PROGRAM F32_InterimPrinter
VAR
END_VAR

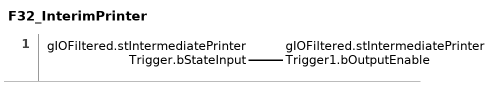
// NETWORK 1
gIOFiltered.stIntermediatePrinterTrigger1.bOutputEnable := gIOFiltered.stIntermediatePrinterTrigger.bStateInput;

END_PROGRAM

(* stored: Version 1.1.0.1
   POU F32_InterimPrinter: Id {b25978ef-63de-464c-bc94-2d79b0d8bd85}, SpecialFunc None *)
